FUNCTION F_TB_SV2STR : STRING
VAR_INPUT
	SV: REAL;
END_VAR
VAR
	r1: REAL;
	iSV: LINT;
	str: STRING;
END_VAR

// SMC HEBC002-WA10
// sv >= 0 -> '00010'
// sv < 0 -> '-0010'
r1 := SV * 10;
iSV := REAL_TO_LINT(r1);
IF iSV >= 0 THEN
	str := LINT_TO_DECSTR(in:=iSV, iPrecision:=5);
ELSE
	str := CONCAT('', LINT_TO_DECSTR(in:=iSV, iPrecision:=4));	//CONCAT('-', LINT_TO_DECSTR(in:=iSV, iPrecision:=4));	
END_IF
F_TB_SV2STR := str;

END_FUNCTION

(* stored: Version 1.1.0.1, ProductVersion 3.1.4024.12
   POU F_TB_SV2STR: Id {a9f17dcf-3769-4132-997d-cb34da53042b}, SpecialFunc None *)
